FUNCTION_BLOCK FB_Lens IMPLEMENTS I_Lens
VAR
    {attribute 'pytmc' := '
        pv: Delta
        io: i
    '}
    fDelta : LREAL;

    {attribute 'pytmc' := '
        pv: Error
        io: i
    '}
    bError : BOOL;

    {attribute 'pytmc' := '
        pv: f1
        io: i
    '}
    fF1 : LREAL;

    {attribute 'pytmc' := '
        pv: FocalLength
        io: i
    '}
    fFocalLength : LREAL;

    {attribute 'pytmc' := '
        pv: Energy
        io: io
    '}
    fEnergy : LREAL;

    {attribute 'pytmc' := '
        pv: Radius
        io: io
    '}
    fRadius : LREAL;

    {attribute 'pytmc' := '
        pv: Multiplier
        io: io
    '}
    nMultiplier : INT;

    {attribute 'pytmc' := '
        pv: ErrorMsg
        io: i
    '}
    sErrorMsg : T_MaxString;

    {attribute 'pytmc' := 'pv: Material'}
    fbMaterial : FB_Element;
END_VAR


PROPERTY Delta : LREAL
GET
VAR
    fbXRayDelta : FB_XRayDelta;
END_VAR

fbXRayDelta(
    fEnergy := Energy,
    fF1 := f1,
    fDensity := fbMaterial.Density,
    nAtomicNumber := fbMaterial.Protons,
    fAtomicMass := fbMaterial.Mass,
    fDelta =>,
    bError =>,
    sErrorMsg =>
);

IF fbXRayDelta.bError THEN
    bError := TRUE;
    sErrorMsg := fbXRayDelta.sErrorMsg;
ELSE
    fDelta := fbXRayDelta.fDelta;
END_IF

Delta := fDelta;
END_GET
END_PROPERTY


PROPERTY Energy : LREAL
GET

// Check for a negative photon energy.
IF fEnergy < 0.0 THEN
    // If we have an invalid photon energy value, give an error.
    bError := TRUE;
    sErrorMsg := CONCAT('Invalid photon energy value of: [',
        CONCAT(LREAL_TO_STRING(fEnergy),
        ']. Must be greater than or equal to 0.'));
END_IF

Energy := fEnergy;
END_GET
SET

fEnergy := Energy;
END_SET
END_PROPERTY


PROPERTY Error : BOOL
GET

Error := bError;
END_GET
END_PROPERTY


PROPERTY ErrorMsg : T_MaxString
GET

ErrorMsg := sErrorMsg;
END_GET
END_PROPERTY


PROPERTY f1 : LREAL
GET

GVL_Physics.fbScatteringFactors(
     sTableName := fbMaterial.Name,
     fEnergyEV := Energy,
     f1 =>,
     bError =>,
     bFound =>,
     bDone =>,
     fTableLookupLow =>,
     fTableLookupHigh =>
);

// Check for an error in retrieving the scattering factor.
IF GVL_Physics.fbScatteringFactors.bDone THEN
    IF GVL_Physics.fbScatteringFactors.bError THEN
        bError := TRUE;
        IF GVL_Physics.fbScatteringFactors.bFound THEN
            // Done but not found and had an error meaning there is no table for the name provided.
            sErrorMsg := CONCAT('The element name provided: [',
                CONCAT(fbMaterial.Name,
                '] does not have a scattering lookup table defined for it.'));
        ELSE
            // Done and found but had an error meaning the table data is flawed.
            sErrorMsg := CONCAT('Detected that the table for the provided element name [',
                CONCAT(fbMaterial.Name,
                '] is not strictly increasing in photon energy with row number. The table is malformed.'));
        END_IF
    ELSIF GVL_Physics.fbScatteringFactors.bFound THEN
        // Done and found and no error meaning we got a valid f1 scattering factor.
        fF1 := GVL_Physics.fbScatteringFactors.f1;
    ELSE
        // Done and no internal error but not found meaning the photon energy exceeds the bounds of our table.
        bError := TRUE;
        IF fEnergy < GVL_Physics.fbScatteringFactors.fTableLookupLow THEN
            sErrorMsg := CONCAT('The photon energy [',
                CONCAT(LREAL_TO_STRING(Energy),
                CONCAT(' eV] provided is lower than the scattering factor lookup table has data for. The lowest table value is: [',
                CONCAT(LREAL_TO_STRING(GVL_Physics.fbScatteringFactors.fTableLookupLow),
                ' eV]'))));
        ELSIF fEnergy > GVL_Physics.fbScatteringFactors.fTableLookupHigh THEN
            sErrorMsg := CONCAT('The photon energy [',
                CONCAT(LREAL_TO_STRING(fEnergy),
                CONCAT(' eV] provided is higher than the scattering factor lookup table has data for. The highest table value is: [',
                CONCAT(LREAL_TO_STRING(GVL_Physics.fbScatteringFactors.fTableLookupHigh),
                ' eV]'))));
        END_IF
    END_IF
END_IF

f1 := fF1;
END_GET
END_PROPERTY


PROPERTY FocalLength : LREAL
GET
VAR
    fbCalcFocalLengthSingleLens : FB_CalcFocalLengthSingleLens;
END_VAR

fbCalcFocalLengthSingleLens(
    fDelta := Delta,
    fRadius := Radius,
    fFocalLength =>,
    bError =>,
    sErrorMsg =>
);

IF fbCalcFocalLengthSingleLens.bError THEN
    bError := TRUE;
    sErrorMsg := fbCalcFocalLengthSingleLens.sErrorMsg;
ELSE
    fFocalLength := fbCalcFocalLengthSingleLens.fFocalLength;
END_IF

FocalLength := fFocalLength;
END_GET
END_PROPERTY


PROPERTY Material : FB_Element
GET

Material := fbMaterial;
END_GET
SET

fbMaterial := Material;
END_SET
END_PROPERTY


PROPERTY Multiplier : INT
GET

// Check for an invalid multiplier.
IF nMultiplier <= 0 THEN
    // If we have an invalid multiplier value, give an error.
    bError := TRUE;
    sErrorMsg := CONCAT('Invalid multiplier value of: [',
        CONCAT(LREAL_TO_STRING(nMultiplier),
        ']. Must be greater than 0.'));
END_IF

Multiplier := nMultiplier;
END_GET
SET

nMultiplier := Multiplier;
END_SET
END_PROPERTY


PROPERTY Radius : LREAL
GET

// Check for an invalid radius of curvature.
IF fRadius <= 0.0 THEN
    // If we have an invalid radius value, give an error.
    bError := TRUE;
    sErrorMsg := CONCAT('Invalid radius of curvature value of: [',
        CONCAT(LREAL_TO_STRING(fRadius),
        ']. Must be greater than 0.'));
END_IF

Radius := fRadius;
END_GET
SET

fRadius := Radius;
END_SET
END_PROPERTY

END_FUNCTION_BLOCK

(* stored: Version 1.1.0.1, ProductVersion 3.1.4022.18
   POU FB_Lens: Id {4a31c30d-ca3e-4cb7-bedc-d5a5413a2a83}, SpecialFunc None
   Property Delta: Id {953307c9-701a-489d-bb16-3ab7bbcd9dab}
   Get Get: Id {9dc56aac-ad27-4ad2-8159-763355bf3777}
   Property Energy: Id {241c4d6d-a08b-4aaf-94a8-16094f2379be}
   Get Get: Id {e154584a-9896-4183-8b97-09943c7dafe4}
   Set Set: Id {3f4d6ab6-fe4a-4712-841e-47e0eefbdb7b}
   Property Error: Id {6d034299-a490-4dad-8873-8a89e1e2c6fa}
   Get Get: Id {c876d34c-4b2f-410b-80ff-69b10dc64f40}
   Property ErrorMsg: Id {02a33bd4-467c-45af-a0ce-3613e5502284}
   Get Get: Id {c522b1a1-236a-4345-a7bc-997738e3275d}
   Property f1: Id {2300ba17-2d98-4b84-ad62-0f58fef3ee00}
   Get Get: Id {44a05807-f5cd-4918-9627-89f90a4b9efa}
   Property FocalLength: Id {dc08c5d9-57d2-4db2-b9d6-81a3f093c3a7}
   Get Get: Id {90f636aa-67bc-466a-8b61-824902ec7a95}
   Property Material: Id {23cb63db-07d0-4116-ab90-923d7879ff4f}
   Get Get: Id {da72f42c-3df6-4714-a29b-6bc43cdfb118}
   Set Set: Id {6ce73d05-2462-44ce-8e89-d88b495103ed}
   Property Multiplier: Id {98fc8c2e-c6d7-409d-b4a9-db30074d0ee6}
   Get Get: Id {a9863f33-2967-4a47-beed-f3a5c59bf8dd}
   Set Set: Id {d57ed44a-0934-4031-a8c3-de43028beb6a}
   Property Radius: Id {3104537e-912b-4e56-9c53-aa6b3018a730}
   Get Get: Id {cccdf607-9ba6-4470-aaaa-400a0e58cdb1}
   Set Set: Id {0fb7c51b-5b18-405a-8d02-c569f9ba7a4c} *)
